(* CODESYS project TrafficLight.project

Project tree, tasks and I/O mapping:
  Device : CODESYS Control Win V3, 3S - Smart Software Solutions GmbH, order no. 305021, version 3.5.10.30
    application Application
      libraries: Standard, * (System)
      task MainTask (cyclic, interval t#20ms, priority 1) calls PLC_PRG
      task VISU_TASK (cyclic, interval 100 ms, priority 31) calls VisuElems.Visu_Prg
      program PLC_PRG [FBD]
      function block NormalCycle_FB [ST]
      function block BlinkingYellow_FB [ST]
      visualisation Visualization
  text list GlobalTextList
*)

// Device/Application/PLC_PRG
PROGRAM PLC_PRG
VAR
	NormalCycle_FB_0: NormalCycle_FB;
	Contact1: BOOL;
	CoilRed: BOOL;
	CoilYellow: BOOL;
	CoilGreen: BOOL;
	Error: BOOL;
	BlinkingYellow_FB_0: BlinkingYellow_FB;
	CoilYellow2: BOOL;
END_VAR

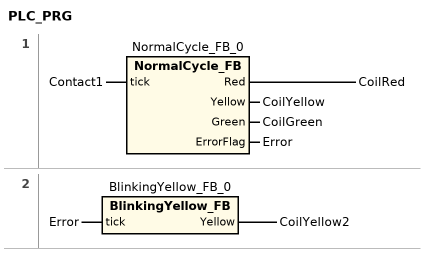
// NETWORK 1
NormalCycle_FB_0(tick := Contact1, Yellow => CoilYellow, Green => CoilGreen, ErrorFlag => Error); // NormalCycle_FB
CoilRed := NormalCycle_FB_0.Red;

// NETWORK 2
BlinkingYellow_FB_0(tick := Error); // BlinkingYellow_FB
CoilYellow2 := BlinkingYellow_FB_0.Yellow;

END_PROGRAM

// Device/Application/NormalCycle_FB
FUNCTION_BLOCK NormalCycle_FB
VAR_INPUT
	tick : BOOL;
END_VAR

VAR_OUTPUT
	Red : BOOL;
	Yellow : BOOL;
	Green : BOOL;
	ErrorFlag : BOOL := FALSE;
END_VAR

VAR
	Counter : INT := 0;
	State : INT := 0;
	Delay : TON;
	
	(*Fake error after set led red 5 time*)
	FakeError: INT := 0;
END_VAR

IF tick = TRUE THEN
	CASE State OF
		0: IF FakeError = 3 THEN (*Fake error triggered after 5 time red*)
				ErrorFlag := TRUE;
				Yellow := FALSE;
				RETURN;
			END_IF
			Red := TRUE;
			Yellow := FALSE;
			Green := FALSE;
			Delay(IN:= NOT Delay.Q, PT:=T#10S);
			IF Delay.Q THEN
				State := 2;
				Counter := Counter + 1;
				FakeError := FakeError + 1;
			END_IF
										
		1:	Yellow := TRUE;
			Red := FALSE;
			Green := FALSE;
			Delay(IN:= NOT Delay.Q, PT:=T#5S);
			IF Delay.Q THEN
				State := 0;
				Counter := Counter + 1;
			END_IF					
					
		2:	Green := TRUE;
			Red := FALSE;
			Yellow := FALSE;
			Delay(IN:= NOT Delay.Q, PT:=T#15S);
			IF Delay.Q THEN
				State := 1;
				Counter := Counter + 1;
			END_IF
		
		ELSE
			ErrorFlag := TRUE;
			Green := FALSE;
			Yellow := FALSE;
			Red := FALSE;
			State := 4;
	
		END_CASE	
	
ELSE
	(*Reset*)
	Green := FALSE;
	Yellow := FALSE;
	Red := FALSE;
	State := 0;
	Counter := 0;
	FakeError := 0;
	ErrorFlag := FALSE;
END_IF

END_FUNCTION_BLOCK

// Device/Application/BlinkingYellow_FB
FUNCTION_BLOCK BlinkingYellow_FB
VAR_INPUT
	tick : BOOL;
END_VAR
	
VAR_OUTPUT
	Yellow : BOOL;
END_VAR

VAR
	State : INT := 4;
	Delay : TON;
END_VAR

IF tick THEN
	CASE State OF
		4 :	Yellow := TRUE;
			delay(IN := NOT delay.Q, PT := T#3S);
			IF delay.Q THEN
				state := 5;
			END_IF
		
		5:	Yellow := FALSE;
			delay(IN := NOT delay.Q, PT := T#3S);
			IF delay.Q THEN
				state := 4;
			END_IF
	END_CASE
END_IF

END_FUNCTION_BLOCK

// Device/Application/Visualization
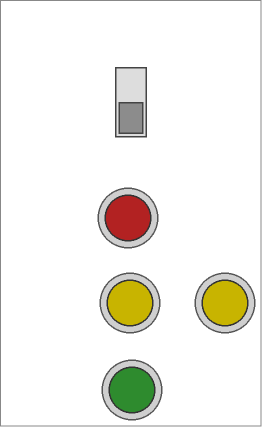
VISUALIZATION Visualization  // 262x427
    Lamp1 (93,183 70x70), variable: PLC_PRG.CoilRed, style: Lamp-Lamp1-Red
    Lamp1 (95,268 70x70), variable: PLC_PRG.CoilYellow, style: Lamp-Lamp1-Yellow
    Lamp1 (97,355 70x70), variable: PLC_PRG.CoilGreen, style: Lamp-Lamp1-Green
    DipSwitch (96,67 70x70), variable: PLC_PRG.Contact1, behaviour: TOGGLE, style: Switch-DipSwitch-Gray
    Lamp1 (190,268 70x70), variable: PLC_PRG.CoilYellow2, style: Lamp-Lamp1-Yellow
END_VISUALIZATION
